(* PLC project Scenario_4b, Beckhoff Automation GmbH TwinCAT PLC Control 3.5.8.40 *)
(* stored: creationDateTime 2017-07-24T10:06:21.7701888, modificationDateTime 2017-07-24T10:06:21.774189 *)

PROGRAM MAIN
                                            VAR
                                            PPU : PPU;

                                            //WPType
                                            //Stack WPType
                                            Stack_WPType_Black : BOOL;
                                            Stack_WPType_White : BOOL;
                                            Stack_WPType_Metallic : BOOL;
                                            //Crane WPType
                                            Crane_WPType_Black : BOOL;
                                            Crane_WPType_White : BOOL;
                                            Crane_WPType_Metallic : BOOL;
                                            //Stamp WPType
                                            Stamp_WPType_Black : BOOL;
                                            Stamp_WPType_White : BOOL;
                                            Stamp_WPType_Metallic : BOOL;

                                            //Free Signale for follow plant section
                                            //Stack
                                            Stack_WPProvided : BOOL;
                                            //Crane
                                            Crane_Allow_Stamp_to_Operate : BOOL;
                                            Crane_PickedUpStackWP : BOOL;
                                            //Stamp
                                            Stamp_IsStamping : BOOL;
                                            Stamp_WPAvailable : BOOL;
                                            Stamp_AutomaticExecuteCompleted : BOOL;

                                            END_VAR

                                    PPU();
                                        PPU.Stack();
                                        PPU.Crane();
                                        PPU.Stamp();


                                        //WPType
                                        //Stack WPType
                                        Stack_WPType_Black := PPU.Stack.WPType_Black;
                                        Stack_WPType_Metallic := PPU.Stack.WPType_Metallic;
                                        //Crane WPType
                                        Crane_WPType_Black := PPU.Crane.WPType_Black;
                                        Crane_WPType_Metallic := PPU.Crane.WPType_Metallic;
                                        //Stamp WPType
                                        Stamp_WPType_Black := PPU.Stamp.WPType_Black;
                                        Stamp_WPType_Metallic := PPU.Stamp.WPType_Metallic;

                                        //Free Signale for follow plant section
                                        //Stack
                                        Stack_WPProvided := PPU.Stack.WPProvided;
                                        //Crane
                                        Crane_Allow_Stamp_to_Operate := PPU.Crane.Stamp_AllowedToOperate;
                                        Crane_PickedUpStackWP := PPU.Crane.Table.AtStack.DI_SwitchTrue AND
                                        PPU.Crane.WPPickedUp;
                                        //Stamp
                                        Stamp_IsStamping := PPU.Stamp.IsStamping;
                                        Stamp_WPAvailable := PPU.Stamp.WPAvailable.DI_SwitchTrue;
                                        Stamp_AutomaticExecuteCompleted := PPU.Stamp.AutomaticExecuteCompleted;
                                    
                                
END_PROGRAM

FUNCTION_BLOCK BistableCylinder
                                            VAR_INPUT
                                            END_VAR
                                            VAR_OUTPUT
                                            //Software
                                            Extended : BOOL;
                                            Retracted : BOOL;
                                            END_VAR
                                            VAR
                                            //Hardware
                                            DI_Extended AT %I* : BOOL;
                                            DI_Retracted AT %I* : BOOL;
                                            DO_Extend AT %Q* : BOOL;
                                            DO_Retract AT %Q* : BOOL;
                                            END_VAR

                                    
                                

ACTION ACT_Extend:
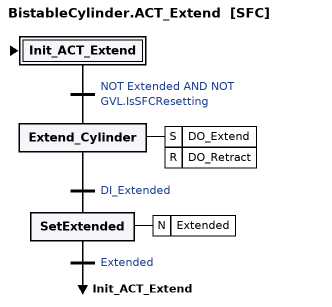
INITIAL_STEP Init_ACT_Extend:
END_STEP
TRANSITION FROM Init_ACT_Extend TO Extend_Cylinder
  := NOT Extended AND NOT GVL.IsSFCResetting;
END_TRANSITION
STEP Extend_Cylinder:
  DO_Extend(S);
  DO_Retract(R);
END_STEP
TRANSITION FROM Extend_Cylinder TO SetExtended
  := DI_Extended;
END_TRANSITION
STEP SetExtended:
  Extended(N);
END_STEP
TRANSITION FROM SetExtended TO Init_ACT_Extend
  := Extended;
END_TRANSITION
END_ACTION

ACTION ACT_Retract:
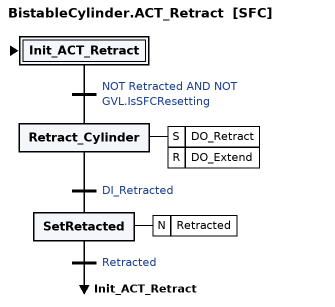
INITIAL_STEP Init_ACT_Retract:
END_STEP
TRANSITION FROM Init_ACT_Retract TO Retract_Cylinder
  := NOT Retracted AND NOT GVL.IsSFCResetting;
END_TRANSITION
STEP Retract_Cylinder:
  DO_Retract(S);
  DO_Extend(R);
END_STEP
TRANSITION FROM Retract_Cylinder TO SetRetacted
  := DI_Retracted;
END_TRANSITION
STEP SetRetacted:
  Retracted(N);
END_STEP
TRANSITION FROM SetRetacted TO Init_ACT_Retract
  := Retracted;
END_TRANSITION
END_ACTION
END_FUNCTION_BLOCK

FUNCTION_BLOCK InductiveSensor
                                            VAR_INPUT
                                            END_VAR
                                            VAR_OUTPUT
                                            END_VAR
                                            VAR
                                            //Hardware
                                            DI_WPMetallic AT %I* : BOOL;
                                            END_VAR

                                    
                                
END_FUNCTION_BLOCK

FUNCTION_BLOCK MicroSwitch
                                            VAR_INPUT
                                            END_VAR
                                            VAR_OUTPUT
                                            END_VAR
                                            VAR
                                            //Hardware
                                            DI_SwitchTrue AT %I* : BOOL;
                                            END_VAR

                                    
                                
END_FUNCTION_BLOCK

FUNCTION_BLOCK InductiveSwitch
                                            VAR_INPUT
                                            END_VAR
                                            VAR_OUTPUT
                                            END_VAR
                                            VAR
                                            //Hardware
                                            DI_InductiveSwitchTrue AT %I* : BOOL;
                                            END_VAR

                                    
                                
END_FUNCTION_BLOCK

FUNCTION_BLOCK MonostableCylinder
                                            VAR_INPUT
                                            END_VAR
                                            VAR_OUTPUT
                                            //Software
                                            Extended : BOOL;
                                            Retracted : BOOL;
                                            END_VAR
                                            VAR
                                            //Hardware
                                            DI_Extended AT %I* : BOOL;
                                            DI_Retracted AT %I* : BOOL;
                                            DO_Extend AT %Q* : BOOL;
                                            END_VAR

                                    
                                

ACTION ACT_Extend:
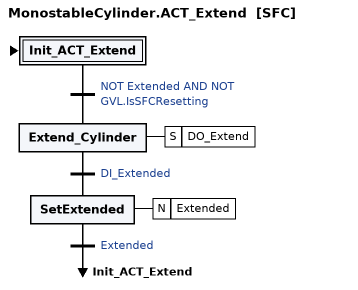
INITIAL_STEP Init_ACT_Extend:
END_STEP
TRANSITION FROM Init_ACT_Extend TO Extend_Cylinder
  := NOT Extended AND NOT GVL.IsSFCResetting;
END_TRANSITION
STEP Extend_Cylinder:
  DO_Extend(S);
END_STEP
TRANSITION FROM Extend_Cylinder TO SetExtended
  := DI_Extended;
END_TRANSITION
STEP SetExtended:
  Extended(N);
END_STEP
TRANSITION FROM SetExtended TO Init_ACT_Extend
  := Extended;
END_TRANSITION
END_ACTION

ACTION ACT_Retract:
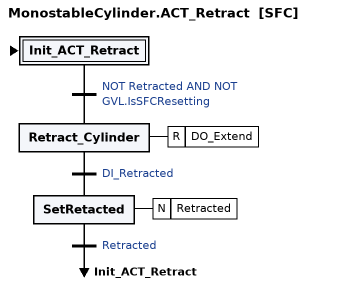
INITIAL_STEP Init_ACT_Retract:
END_STEP
TRANSITION FROM Init_ACT_Retract TO Retract_Cylinder
  := NOT Retracted AND NOT GVL.IsSFCResetting;
END_TRANSITION
STEP Retract_Cylinder:
  DO_Extend(R);
END_STEP
TRANSITION FROM Retract_Cylinder TO SetRetacted
  := DI_Retracted;
END_TRANSITION
STEP SetRetacted:
  Retracted(N);
END_STEP
TRANSITION FROM SetRetacted TO Init_ACT_Retract
  := Retracted;
END_TRANSITION
END_ACTION
END_FUNCTION_BLOCK

FUNCTION_BLOCK Motor
                                            VAR_INPUT
                                            END_VAR
                                            VAR_OUTPUT
                                            //Software
                                            Stopped : BOOL;
                                            TurningClockwise : BOOL;
                                            TurningCounterclockwise : BOOL;
                                            END_VAR
                                            VAR
                                            //Hardware
                                            DO_TurnClockwise AT %Q* : BOOL;
                                            DO_TurnCounterclockwise AT %Q* : BOOL;
                                            END_VAR

                                    
                                

ACTION ACT_Stop:
                                            DO_TurnClockwise := FALSE;
                                                DO_TurnCounterclockwise := FALSE;

                                                Stopped := TRUE;
                                                TurningClockwise := FALSE;
                                                TurningCounterclockwise := FALSE;
                                            
                                        
END_ACTION

ACTION ACT_TurnClockwise:
                                            DO_TurnClockwise := TRUE;
                                                DO_TurnCounterclockwise := FALSE;

                                                Stopped := FALSE;
                                                TurningClockwise := TRUE;
                                                TurningCounterclockwise := FALSE;
                                            
                                        
END_ACTION

ACTION ACT_TurnCounterclockwise:
                                            DO_TurnClockwise := FALSE;
                                                DO_TurnCounterclockwise := TRUE;

                                                Stopped := FALSE;
                                                TurningClockwise := FALSE;
                                                TurningCounterclockwise := TRUE;
                                            
                                        
END_ACTION
END_FUNCTION_BLOCK

FUNCTION_BLOCK OperationPanel
                                            VAR_INPUT
                                            END_VAR
                                            VAR_OUTPUT
                                            //Software
                                            EmergencyStop : BOOL;
                                            StartButton : BOOL;
                                            ManuelMode : BOOL;
                                            END_VAR
                                            VAR
                                            //Hardware
                                            DI_StartButton AT %I* : BOOL;
                                            DI_ManuelButton AT %I* : BOOL;
                                            DI_EmergencyStop AT %I* : BOOL;
                                            DO_LampGreen AT %Q* : BOOL;
                                            DO_LampWhite AT %Q* : BOOL;
                                            END_VAR

                                    EmergencyStop := NOT DI_EmergencyStop;
                                        StartButton := DI_StartButton;
                                        ManuelMode := DI_ManuelButton;
                                    
                                

ACTION ACT_TurnLampGreen_Off:
                                            DO_LampGreen := FALSE;
                                        
END_ACTION

ACTION ACT_TurnLampGreen_On:
                                            DO_LampGreen := TRUE;
                                        
END_ACTION

ACTION ACT_TurnLampWhite_Off:
                                            DO_LampWhite:=FALSE;
                                        
END_ACTION

ACTION ACT_TurnLampWhite_On:
                                            DO_LampWhite:=TRUE;
                                        
END_ACTION
END_FUNCTION_BLOCK

FUNCTION_BLOCK ProportionalValve
                                            VAR_INPUT
                                            //Hardware
                                            AO_SetPressure AT %Q* : INT;
                                            END_VAR
                                            VAR_OUTPUT
                                            END_VAR
                                            VAR
                                            END_VAR

                                    
                                
END_FUNCTION_BLOCK

FUNCTION_BLOCK TurningTable
                                            VAR_INPUT
                                            END_VAR
                                            VAR_OUTPUT
                                            END_VAR
                                            VAR
                                            //Hardware
                                            Motor : Motor;
                                            AtStack : MicroSwitch;
                                            AtRamp : MicroSwitch;
                                            AtStamp : MicroSwitch;
                                            AtStackInd : InductiveSwitch;
                                            AtRampInd : InductiveSwitch;
                                            AtStampInd : InductiveSwitch;

                                            END_VAR

                                    
                                
END_FUNCTION_BLOCK

FUNCTION_BLOCK VacuumGripper
                                            VAR_INPUT
                                            //Hardware
                                            Valve : Valve;
                                            VacuumSwitch : VacuumSwitch;
                                            END_VAR
                                            VAR_OUTPUT
                                            //Software
                                            Intaken : BOOL;
                                            Released : BOOL;
                                            END_VAR
                                            VAR
                                            END_VAR

                                    
                                

ACTION ACT_Intake:
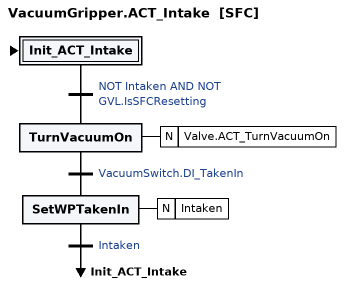
INITIAL_STEP Init_ACT_Intake:
END_STEP
TRANSITION FROM Init_ACT_Intake TO TurnVacuumOn
  := NOT Intaken AND NOT GVL.IsSFCResetting;
END_TRANSITION
STEP TurnVacuumOn:
  Valve.ACT_TurnVacuumOn(N);
END_STEP
TRANSITION FROM TurnVacuumOn TO SetWPTakenIn
  := VacuumSwitch.DI_TakenIn;
END_TRANSITION
STEP SetWPTakenIn:
  Intaken(N);
END_STEP
TRANSITION FROM SetWPTakenIn TO Init_ACT_Intake
  := Intaken;
END_TRANSITION
END_ACTION

ACTION ACT_Release:
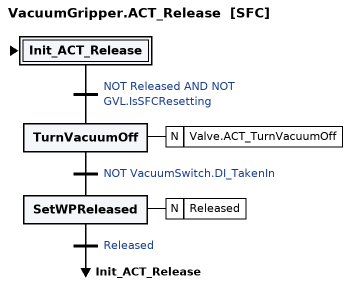
INITIAL_STEP Init_ACT_Release:
END_STEP
TRANSITION FROM Init_ACT_Release TO TurnVacuumOff
  := NOT Released AND NOT GVL.IsSFCResetting;
END_TRANSITION
STEP TurnVacuumOff:
  Valve.ACT_TurnVacuumOff(N);
END_STEP
TRANSITION FROM TurnVacuumOff TO SetWPReleased
  := NOT VacuumSwitch.DI_TakenIn;
END_TRANSITION
STEP SetWPReleased:
  Released(N);
END_STEP
TRANSITION FROM SetWPReleased TO Init_ACT_Release
  := Released;
END_TRANSITION
END_ACTION
END_FUNCTION_BLOCK

FUNCTION_BLOCK VacuumSwitch
                                            VAR_INPUT
                                            END_VAR
                                            VAR_OUTPUT
                                            END_VAR
                                            VAR
                                            //Hardware
                                            DI_TakenIn AT %I* : BOOL;
                                            END_VAR

                                    
                                
END_FUNCTION_BLOCK

FUNCTION_BLOCK Valve
                                            VAR_INPUT
                                            END_VAR
                                            VAR_OUTPUT
                                            END_VAR
                                            VAR
                                            //Hardware
                                            DO_VacuumOn AT %Q* : BOOL;
                                            END_VAR

                                    
                                

ACTION ACT_TurnVacuumOff:
                                            DO_VacuumOn := FALSE;
                                        
END_ACTION

ACTION ACT_TurnVacuumOn:
                                            DO_VacuumOn := TRUE;
                                        
END_ACTION
END_FUNCTION_BLOCK

FUNCTION_BLOCK Crane
                                            VAR_INPUT
                                            //Hardware
                                            LiftingCylinder : MonostableCylinder;
                                            Gripper : VacuumGripper;
                                            Table : TurningTable;
                                            //Software
                                            InitCompleted : BOOL;
                                            AutomaticExecuteCompleted : BOOL;
                                            Stamp_AllowedToOperate : BOOL;
                                            Stamp_WPStamped : BOOL;
                                            SoftwareEmergency : BOOL;
                                            EmergencyHandled : BOOL;
                                            SFCReset : BOOL; //Only for SFC implementation
                                            END_VAR
                                            VAR_OUTPUT
                                            //Software
                                            WPPickedUp : BOOL;
                                            WPPutDown : BOOL;
                                            ReachedStack : BOOL;
                                            ReachedRamp : BOOL;
                                            ReachedStamp : BOOL;
                                            WPType_Black : BOOL;
                                            WPType_Metallic : BOOL;
                                            END_VAR
                                            VAR
                                            //Hardware
                                            CraneSpeed AT %Q* : INT;

                                            //Software
                                            Timer : TON;
                                            Check_Stack_WPProvided : BOOL;
                                            Check_Stack_WPType_Black : BOOL;
                                            Check_Stack_WPType_Metallic : BOOL;
                                            Check_Stamp_IsStamping : BOOL;
                                            Check_Stamp_WPAvailable : BOOL;
                                            Check_Stamp_AutomaticExecuteCompleted : BOOL;
                                            END_VAR

                                    Check_Stack_WPProvided :=
                                        Main.Stack_WPProvided;
                                        Check_Stack_WPType_Black := Main.Stack_WPType_Black;
                                        Check_Stack_WPType_Metallic := Main.Stack_WPType_Metallic;
                                        Check_Stamp_IsStamping := Main.Stamp_IsStamping;
                                        Check_Stamp_WPAvailable := Main.Stamp_WPAvailable;
                                        Check_Stamp_AutomaticExecuteCompleted := Main.Stamp_AutomaticExecuteCompleted;
                                    
                                

ACTION Reset_StampAllowedToOperate:
                                            Stamp_AllowedToOperate :=
                                                FALSE;
                                            
                                        
END_ACTION

ACTION Reset_Timer:
                                            Timer(IN:=FALSE);
                                        
END_ACTION

ACTION Reset_Variables:
                                            InitCompleted := FALSE;
                                                AutomaticExecuteCompleted := FALSE;
                                                Stamp_AllowedToOperate := FALSE;

                                                WPPickedUp := FALSE;
                                                WPPutDown := FALSE;
                                                ReachedStack := FALSE;
                                                ReachedRamp := FALSE;
                                                ReachedStamp := FALSE;
                                                WPType_Black := FALSE;
                                                WPType_Metallic := FALSE;
                                            
                                        
END_ACTION

ACTION Set_StampAllowedToOperate:
                                            Stamp_AllowedToOperate :=
                                                TRUE;
                                            
                                        
END_ACTION

ACTION Set_Timer50ms:
                                            Timer(IN:=TRUE, PT:=T#50MS);
                                            
                                        
END_ACTION

ACTION Set_WPTypeEqualsStack:
                                            
                                                WPType_Black:=Main.Stack_WPType_Black;
                                                WPType_Metallic:=Main.Stack_WPType_Metallic;
                                            
                                        
END_ACTION

ACTION Set_WPTypeEqualsStamp:
                                            
                                                WPType_Black:=Main.Stamp_WPType_Black;
                                                WPType_Metallic:=Main.Stamp_WPType_Metallic;
                                            
                                        
END_ACTION

ACTION TurnClockwise_AND_Timer8000ms:
                                            Table.Motor.ACT_TurnClockwise();
                                                Timer(IN:=TRUE, PT:=T#8000MS);
                                            
                                        
END_ACTION

ACTION TurnCounterclockwise_AND_Timer8000ms:
                                            
                                                Table.Motor.ACT_TurnCounterclockwise();
                                                Timer(IN:=TRUE, PT:=T#8000MS);
                                            
                                        
END_ACTION

ACTION TurnVacuumOn_AND_Timer2000ms:
                                            Gripper.ACT_Intake();
                                                Timer(IN:=TRUE, PT:=T#2000MS);
                                            
                                        
END_ACTION

ACTION ACT_MoveToRamp:
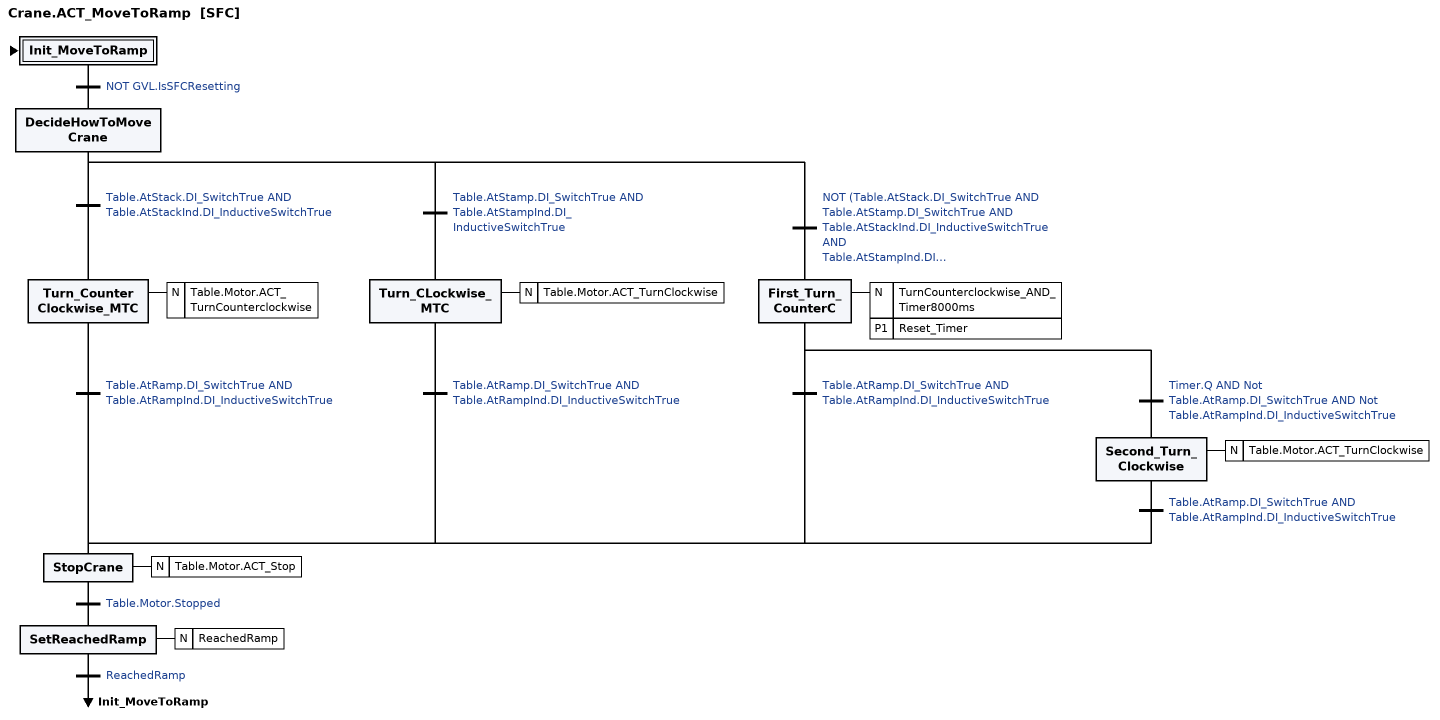
INITIAL_STEP Init_MoveToRamp:
END_STEP
TRANSITION FROM Init_MoveToRamp TO DecideHowToMoveCrane
  := NOT GVL.IsSFCResetting;
END_TRANSITION
STEP DecideHowToMoveCrane:
END_STEP
TRANSITION FROM DecideHowToMoveCrane TO Turn_CounterClockwise_MTC
  := Table.AtStack.DI_SwitchTrue AND
                                                    Table.AtStackInd.DI_InductiveSwitchTrue;
END_TRANSITION
TRANSITION FROM DecideHowToMoveCrane TO Turn_CLockwise_MTC
  := Table.AtStamp.DI_SwitchTrue AND
                                                    Table.AtStampInd.DI_InductiveSwitchTrue;
END_TRANSITION
TRANSITION FROM DecideHowToMoveCrane TO First_Turn_CounterC
  := NOT (Table.AtStack.DI_SwitchTrue AND
                                                    Table.AtStamp.DI_SwitchTrue AND
                                                    Table.AtStackInd.DI_InductiveSwitchTrue AND
                                                    Table.AtStampInd.DI_InductiveSwitchTrue);
END_TRANSITION
STEP Turn_CounterClockwise_MTC:
  Table.Motor.ACT_TurnCounterclockwise(N);
END_STEP
TRANSITION FROM Turn_CounterClockwise_MTC TO StopCrane
  := Table.AtRamp.DI_SwitchTrue AND
                                                    Table.AtRampInd.DI_InductiveSwitchTrue;
END_TRANSITION
STEP Turn_CLockwise_MTC:
  Table.Motor.ACT_TurnClockwise(N);
END_STEP
TRANSITION FROM Turn_CLockwise_MTC TO StopCrane
  := Table.AtRamp.DI_SwitchTrue AND
                                                    Table.AtRampInd.DI_InductiveSwitchTrue;
END_TRANSITION
STEP First_Turn_CounterC:
  TurnCounterclockwise_AND_Timer8000ms(N);
  Reset_Timer(P1);
END_STEP
TRANSITION FROM First_Turn_CounterC TO StopCrane
  := Table.AtRamp.DI_SwitchTrue AND
                                                    Table.AtRampInd.DI_InductiveSwitchTrue;
END_TRANSITION
TRANSITION FROM First_Turn_CounterC TO Second_Turn_Clockwise
  := Timer.Q AND Not Table.AtRamp.DI_SwitchTrue AND Not
                                                    Table.AtRampInd.DI_InductiveSwitchTrue;
END_TRANSITION
STEP Second_Turn_Clockwise:
  Table.Motor.ACT_TurnClockwise(N);
END_STEP
TRANSITION FROM Second_Turn_Clockwise TO StopCrane
  := Table.AtRamp.DI_SwitchTrue AND
                                                    Table.AtRampInd.DI_InductiveSwitchTrue;
END_TRANSITION
STEP StopCrane:
  Table.Motor.ACT_Stop(N);
END_STEP
TRANSITION FROM StopCrane TO SetReachedRamp
  := Table.Motor.Stopped;
END_TRANSITION
STEP SetReachedRamp:
  ReachedRamp(N);
END_STEP
TRANSITION FROM SetReachedRamp TO Init_MoveToRamp
  := ReachedRamp;
END_TRANSITION
END_ACTION

ACTION ACT_MoveToStack:
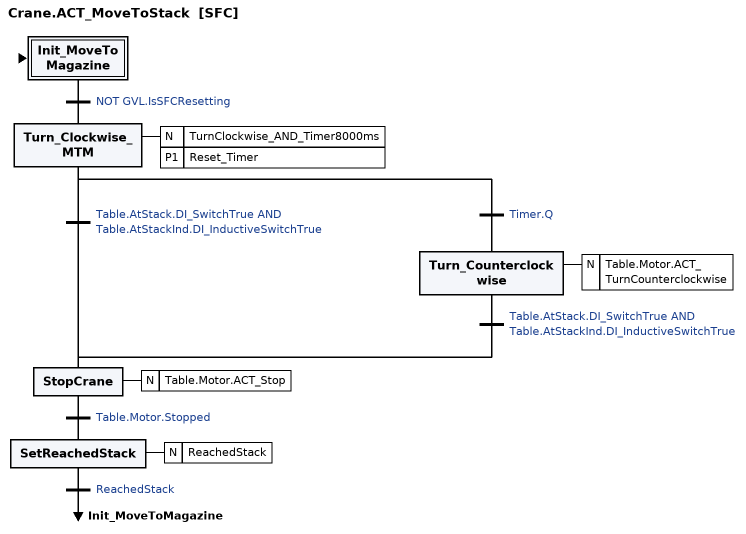
INITIAL_STEP Init_MoveToMagazine:
END_STEP
TRANSITION FROM Init_MoveToMagazine TO Turn_Clockwise_MTM
  := NOT GVL.IsSFCResetting;
END_TRANSITION
STEP Turn_Clockwise_MTM:
  TurnClockwise_AND_Timer8000ms(N);
  Reset_Timer(P1);
END_STEP
TRANSITION FROM Turn_Clockwise_MTM TO StopCrane
  := Table.AtStack.DI_SwitchTrue AND
                                                    Table.AtStackInd.DI_InductiveSwitchTrue;
END_TRANSITION
TRANSITION FROM Turn_Clockwise_MTM TO Turn_Counterclockwise
  := Timer.Q;
END_TRANSITION
STEP Turn_Counterclockwise:
  Table.Motor.ACT_TurnCounterclockwise(N);
END_STEP
TRANSITION FROM Turn_Counterclockwise TO StopCrane
  := Table.AtStack.DI_SwitchTrue AND
                                                    Table.AtStackInd.DI_InductiveSwitchTrue;
END_TRANSITION
STEP StopCrane:
  Table.Motor.ACT_Stop(N);
END_STEP
TRANSITION FROM StopCrane TO SetReachedStack
  := Table.Motor.Stopped;
END_TRANSITION
STEP SetReachedStack:
  ReachedStack(N);
END_STEP
TRANSITION FROM SetReachedStack TO Init_MoveToMagazine
  := ReachedStack;
END_TRANSITION
END_ACTION

ACTION ACT_MoveToStamp:
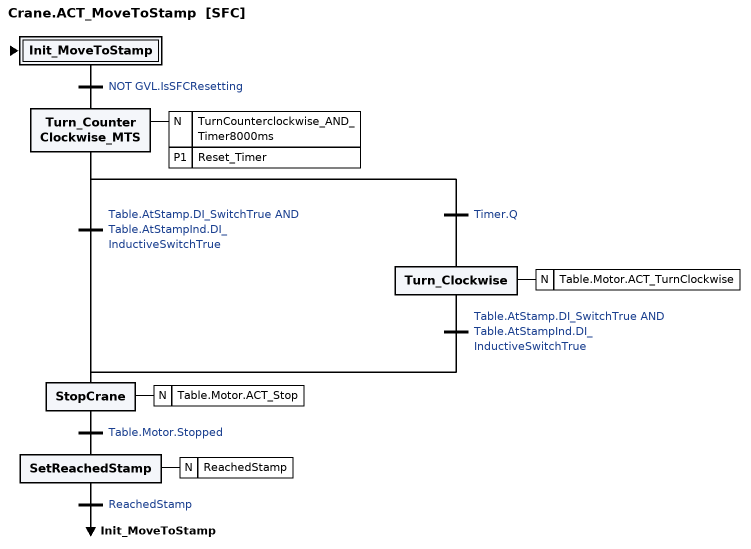
INITIAL_STEP Init_MoveToStamp:
END_STEP
TRANSITION FROM Init_MoveToStamp TO Turn_CounterClockwise_MTS
  := NOT GVL.IsSFCResetting;
END_TRANSITION
STEP Turn_CounterClockwise_MTS:
  TurnCounterclockwise_AND_Timer8000ms(N);
  Reset_Timer(P1);
END_STEP
TRANSITION FROM Turn_CounterClockwise_MTS TO StopCrane
  := Table.AtStamp.DI_SwitchTrue AND
                                                    Table.AtStampInd.DI_InductiveSwitchTrue;
END_TRANSITION
TRANSITION FROM Turn_CounterClockwise_MTS TO Turn_Clockwise
  := Timer.Q;
END_TRANSITION
STEP Turn_Clockwise:
  Table.Motor.ACT_TurnClockwise(N);
END_STEP
TRANSITION FROM Turn_Clockwise TO StopCrane
  := Table.AtStamp.DI_SwitchTrue AND
                                                    Table.AtStampInd.DI_InductiveSwitchTrue;
END_TRANSITION
STEP StopCrane:
  Table.Motor.ACT_Stop(N);
END_STEP
TRANSITION FROM StopCrane TO SetReachedStamp
  := Table.Motor.Stopped;
END_TRANSITION
STEP SetReachedStamp:
  ReachedStamp(N);
END_STEP
TRANSITION FROM SetReachedStamp TO Init_MoveToStamp
  := ReachedStamp;
END_TRANSITION
END_ACTION

ACTION ACT_PickUpWP:
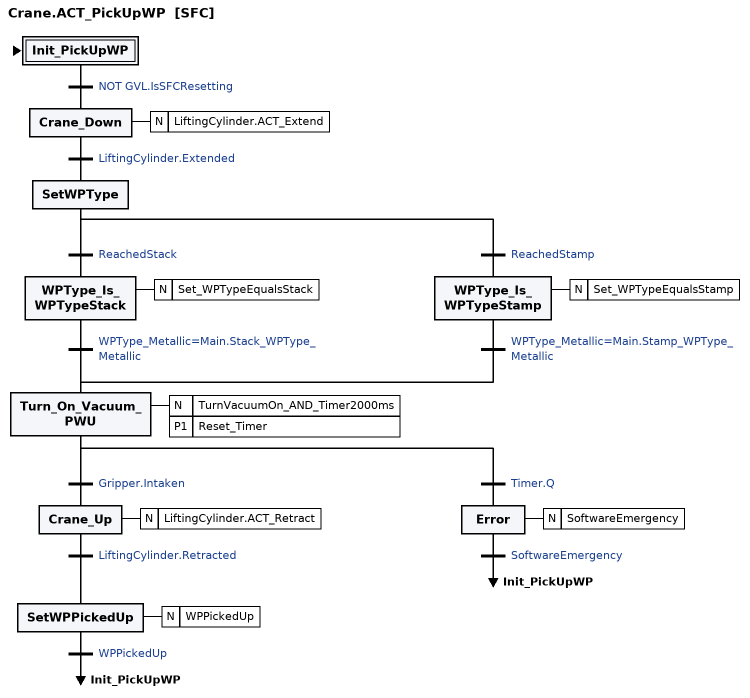
INITIAL_STEP Init_PickUpWP:
END_STEP
TRANSITION FROM Init_PickUpWP TO Crane_Down
  := NOT GVL.IsSFCResetting;
END_TRANSITION
STEP Crane_Down:
  LiftingCylinder.ACT_Extend(N);
END_STEP
TRANSITION FROM Crane_Down TO SetWPType
  := LiftingCylinder.Extended;
END_TRANSITION
STEP SetWPType:
END_STEP
TRANSITION FROM SetWPType TO WPType_Is_WPTypeStack
  := ReachedStack;
END_TRANSITION
TRANSITION FROM SetWPType TO WPType_Is_WPTypeStamp
  := ReachedStamp;
END_TRANSITION
STEP WPType_Is_WPTypeStack:
  Set_WPTypeEqualsStack(N);
END_STEP
TRANSITION FROM WPType_Is_WPTypeStack TO Turn_On_Vacuum_PWU
  := WPType_Metallic=Main.Stack_WPType_Metallic;
END_TRANSITION
STEP WPType_Is_WPTypeStamp:
  Set_WPTypeEqualsStamp(N);
END_STEP
TRANSITION FROM WPType_Is_WPTypeStamp TO Turn_On_Vacuum_PWU
  := WPType_Metallic=Main.Stamp_WPType_Metallic;
END_TRANSITION
STEP Turn_On_Vacuum_PWU:
  TurnVacuumOn_AND_Timer2000ms(N);
  Reset_Timer(P1);
END_STEP
TRANSITION FROM Turn_On_Vacuum_PWU TO Crane_Up
  := Gripper.Intaken;
END_TRANSITION
TRANSITION FROM Turn_On_Vacuum_PWU TO Error
  := Timer.Q;
END_TRANSITION
STEP Crane_Up:
  LiftingCylinder.ACT_Retract(N);
END_STEP
TRANSITION FROM Crane_Up TO SetWPPickedUp
  := LiftingCylinder.Retracted;
END_TRANSITION
STEP Error:
  SoftwareEmergency(N);
END_STEP
TRANSITION FROM Error TO Init_PickUpWP
  := SoftwareEmergency;
END_TRANSITION
STEP SetWPPickedUp:
  WPPickedUp(N);
END_STEP
TRANSITION FROM SetWPPickedUp TO Init_PickUpWP
  := WPPickedUp;
END_TRANSITION
END_ACTION

ACTION ACT_PutDownWP:
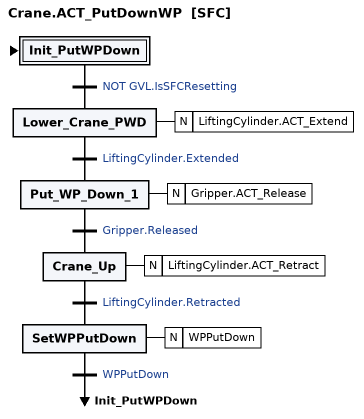
INITIAL_STEP Init_PutWPDown:
END_STEP
TRANSITION FROM Init_PutWPDown TO Lower_Crane_PWD
  := NOT GVL.IsSFCResetting;
END_TRANSITION
STEP Lower_Crane_PWD:
  LiftingCylinder.ACT_Extend(N);
END_STEP
TRANSITION FROM Lower_Crane_PWD TO Put_WP_Down_1
  := LiftingCylinder.Extended;
END_TRANSITION
STEP Put_WP_Down_1:
  Gripper.ACT_Release(N);
END_STEP
TRANSITION FROM Put_WP_Down_1 TO Crane_Up
  := Gripper.Released;
END_TRANSITION
STEP Crane_Up:
  LiftingCylinder.ACT_Retract(N);
END_STEP
TRANSITION FROM Crane_Up TO SetWPPutDown
  := LiftingCylinder.Retracted;
END_TRANSITION
STEP SetWPPutDown:
  WPPutDown(N);
END_STEP
TRANSITION FROM SetWPPutDown TO Init_PutWPDown
  := WPPutDown;
END_TRANSITION
END_ACTION

ACTION ACT_AutomaticExecute:
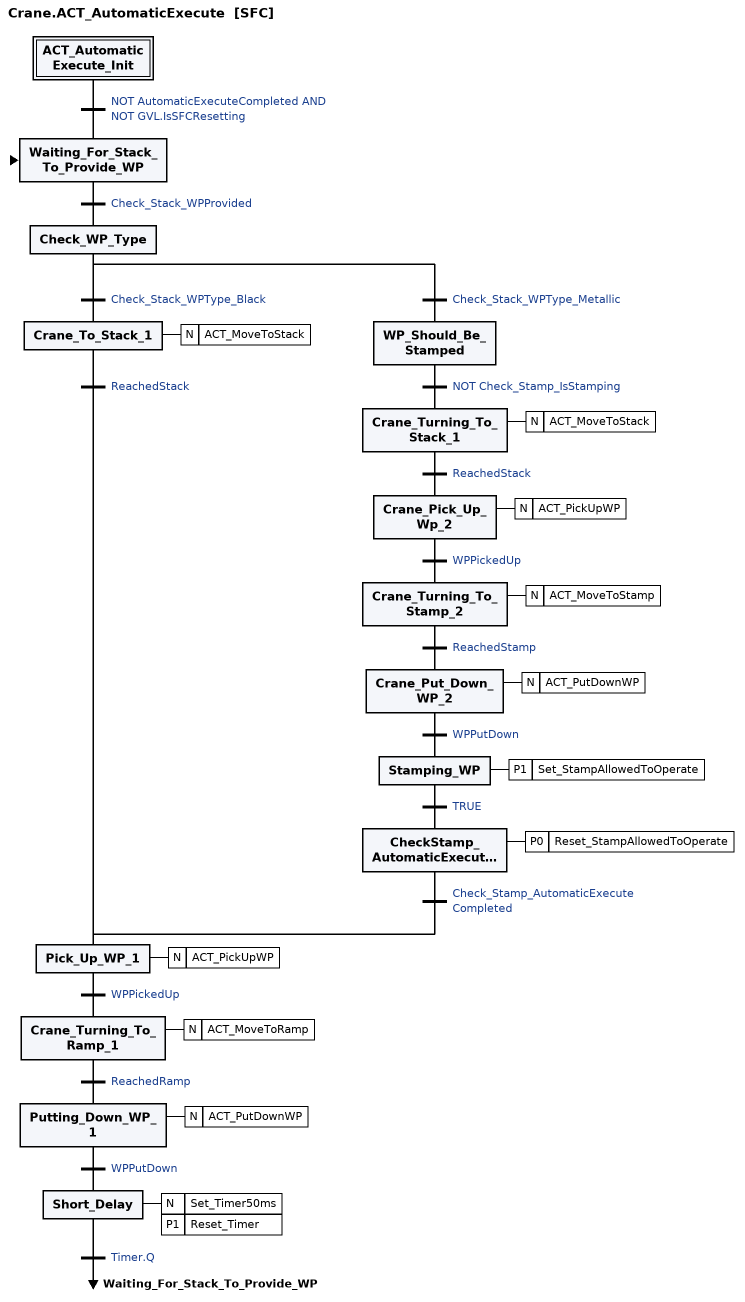
INITIAL_STEP ACT_AutomaticExecute_Init:
END_STEP
TRANSITION FROM ACT_AutomaticExecute_Init TO Waiting_For_Stack_To_Provide_WP
  := NOT AutomaticExecuteCompleted AND NOT GVL.IsSFCResetting;
END_TRANSITION
STEP Waiting_For_Stack_To_Provide_WP:
END_STEP
TRANSITION FROM Waiting_For_Stack_To_Provide_WP TO Check_WP_Type
  := Check_Stack_WPProvided;
END_TRANSITION
STEP Check_WP_Type:
END_STEP
TRANSITION FROM Check_WP_Type TO Crane_To_Stack_1
  := Check_Stack_WPType_Black;
END_TRANSITION
TRANSITION FROM Check_WP_Type TO WP_Should_Be_Stamped
  := Check_Stack_WPType_Metallic;
END_TRANSITION
STEP Crane_To_Stack_1:
  ACT_MoveToStack(N);
END_STEP
TRANSITION FROM Crane_To_Stack_1 TO Pick_Up_WP_1
  := ReachedStack;
END_TRANSITION
STEP Pick_Up_WP_1:
  ACT_PickUpWP(N);
END_STEP
TRANSITION FROM Pick_Up_WP_1 TO Crane_Turning_To_Ramp_1
  := WPPickedUp;
END_TRANSITION
STEP Crane_Turning_To_Ramp_1:
  ACT_MoveToRamp(N);
END_STEP
TRANSITION FROM Crane_Turning_To_Ramp_1 TO Putting_Down_WP_1
  := ReachedRamp;
END_TRANSITION
STEP Putting_Down_WP_1:
  ACT_PutDownWP(N);
END_STEP
TRANSITION FROM Putting_Down_WP_1 TO Short_Delay
  := WPPutDown;
END_TRANSITION
STEP Short_Delay:
  Set_Timer50ms(N);
  Reset_Timer(P1);
END_STEP
TRANSITION FROM Short_Delay TO Waiting_For_Stack_To_Provide_WP
  := Timer.Q;
END_TRANSITION
STEP WP_Should_Be_Stamped:
END_STEP
TRANSITION FROM WP_Should_Be_Stamped TO Crane_Turning_To_Stack_1
  := NOT Check_Stamp_IsStamping;
END_TRANSITION
STEP Crane_Turning_To_Stack_1:
  ACT_MoveToStack(N);
END_STEP
TRANSITION FROM Crane_Turning_To_Stack_1 TO Crane_Pick_Up_Wp_2
  := ReachedStack;
END_TRANSITION
STEP Crane_Pick_Up_Wp_2:
  ACT_PickUpWP(N);
END_STEP
TRANSITION FROM Crane_Pick_Up_Wp_2 TO Crane_Turning_To_Stamp_2
  := WPPickedUp;
END_TRANSITION
STEP Crane_Turning_To_Stamp_2:
  ACT_MoveToStamp(N);
END_STEP
TRANSITION FROM Crane_Turning_To_Stamp_2 TO Crane_Put_Down_WP_2
  := ReachedStamp;
END_TRANSITION
STEP Crane_Put_Down_WP_2:
  ACT_PutDownWP(N);
END_STEP
TRANSITION FROM Crane_Put_Down_WP_2 TO Stamping_WP
  := WPPutDown;
END_TRANSITION
STEP Stamping_WP:
  Set_StampAllowedToOperate(P1);
END_STEP
TRANSITION FROM Stamping_WP TO CheckStamp_AutomaticExecuteCompleted
  := TRUE;
END_TRANSITION
STEP CheckStamp_AutomaticExecuteCompleted:
  Reset_StampAllowedToOperate(P0);
END_STEP
TRANSITION FROM CheckStamp_AutomaticExecuteCompleted TO Pick_Up_WP_1
  := Check_Stamp_AutomaticExecuteCompleted;
END_TRANSITION
END_ACTION

ACTION ACT_EmergencyStop:
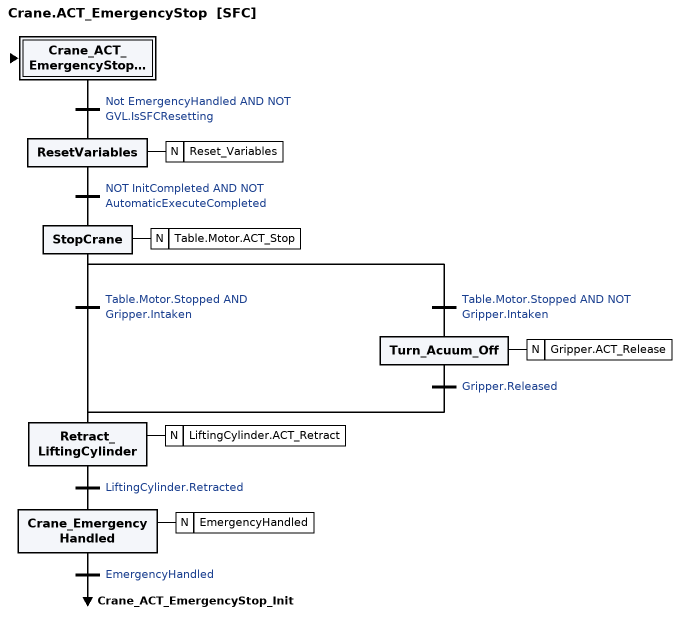
INITIAL_STEP Crane_ACT_EmergencyStop_Init:
END_STEP
TRANSITION FROM Crane_ACT_EmergencyStop_Init TO ResetVariables
  := Not EmergencyHandled AND NOT GVL.IsSFCResetting;
END_TRANSITION
STEP ResetVariables:
  Reset_Variables(N);
END_STEP
TRANSITION FROM ResetVariables TO StopCrane
  := NOT InitCompleted AND NOT AutomaticExecuteCompleted;
END_TRANSITION
STEP StopCrane:
  Table.Motor.ACT_Stop(N);
END_STEP
TRANSITION FROM StopCrane TO Retract_LiftingCylinder
  := Table.Motor.Stopped AND Gripper.Intaken;
END_TRANSITION
TRANSITION FROM StopCrane TO Turn_Acuum_Off
  := Table.Motor.Stopped AND NOT Gripper.Intaken;
END_TRANSITION
STEP Turn_Acuum_Off:
  Gripper.ACT_Release(N);
END_STEP
TRANSITION FROM Turn_Acuum_Off TO Retract_LiftingCylinder
  := Gripper.Released;
END_TRANSITION
STEP Retract_LiftingCylinder:
  LiftingCylinder.ACT_Retract(N);
END_STEP
TRANSITION FROM Retract_LiftingCylinder TO Crane_EmergencyHandled
  := LiftingCylinder.Retracted;
END_TRANSITION
STEP Crane_EmergencyHandled:
  EmergencyHandled(N);
END_STEP
TRANSITION FROM Crane_EmergencyHandled TO Crane_ACT_EmergencyStop_Init
  := EmergencyHandled;
END_TRANSITION
END_ACTION

ACTION ACT_Init:
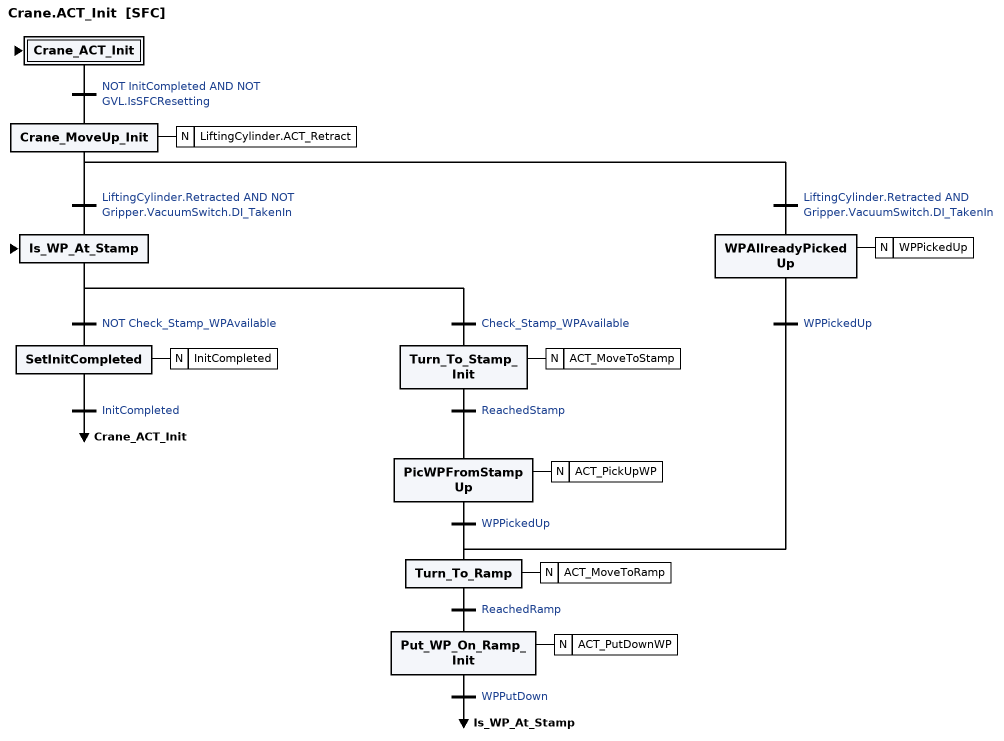
INITIAL_STEP Crane_ACT_Init:
END_STEP
TRANSITION FROM Crane_ACT_Init TO Crane_MoveUp_Init
  := NOT InitCompleted AND NOT GVL.IsSFCResetting;
END_TRANSITION
STEP Crane_MoveUp_Init:
  LiftingCylinder.ACT_Retract(N);
END_STEP
TRANSITION FROM Crane_MoveUp_Init TO Is_WP_At_Stamp
  := LiftingCylinder.Retracted AND NOT
                                                    Gripper.VacuumSwitch.DI_TakenIn;
END_TRANSITION
TRANSITION FROM Crane_MoveUp_Init TO WPAllreadyPickedUp
  := LiftingCylinder.Retracted AND
                                                    Gripper.VacuumSwitch.DI_TakenIn;
END_TRANSITION
STEP WPAllreadyPickedUp:
  WPPickedUp(N);
END_STEP
TRANSITION FROM WPAllreadyPickedUp TO Turn_To_Ramp
  := WPPickedUp;
END_TRANSITION
STEP Turn_To_Ramp:
  ACT_MoveToRamp(N);
END_STEP
TRANSITION FROM Turn_To_Ramp TO Put_WP_On_Ramp_Init
  := ReachedRamp;
END_TRANSITION
STEP Put_WP_On_Ramp_Init:
  ACT_PutDownWP(N);
END_STEP
TRANSITION FROM Put_WP_On_Ramp_Init TO Is_WP_At_Stamp
  := WPPutDown;
END_TRANSITION
STEP Is_WP_At_Stamp:
END_STEP
TRANSITION FROM Is_WP_At_Stamp TO SetInitCompleted
  := NOT Check_Stamp_WPAvailable;
END_TRANSITION
TRANSITION FROM Is_WP_At_Stamp TO Turn_To_Stamp_Init
  := Check_Stamp_WPAvailable;
END_TRANSITION
STEP Turn_To_Stamp_Init:
  ACT_MoveToStamp(N);
END_STEP
TRANSITION FROM Turn_To_Stamp_Init TO PicWPFromStampUp
  := ReachedStamp;
END_TRANSITION
STEP PicWPFromStampUp:
  ACT_PickUpWP(N);
END_STEP
TRANSITION FROM PicWPFromStampUp TO Turn_To_Ramp
  := WPPickedUp;
END_TRANSITION
STEP SetInitCompleted:
  InitCompleted(N);
END_STEP
TRANSITION FROM SetInitCompleted TO Crane_ACT_Init
  := InitCompleted;
END_TRANSITION
END_ACTION
END_FUNCTION_BLOCK

FUNCTION_BLOCK Stack
                                            VAR_INPUT
                                            //Hardware
                                            Seperator : MonostableCylinder;
                                            Panel : OperationPanel;
                                            WPAvailable : MicroSwitch;
                                            InductiveSensor : InductiveSensor;

                                            //Software
                                            StartButton : BOOL;
                                            InitCompleted : BOOL;
                                            AutomaticExecuteCompleted : BOOL;
                                            EmergencyStop : BOOL;
                                            EmergencyHandled : BOOL;
                                            SFCReset : BOOL; //Only for SFC implementation
                                            END_VAR
                                            VAR_OUTPUT
                                            //Software
                                            WPProvided : BOOL;
                                            WPType_Black : BOOL;
                                            WPType_Metallic : BOOL;
                                            END_VAR
                                            VAR
                                            //Software
                                            Timer : TON;
                                            Check_Crane_PickedUpWp : BOOL;
                                            END_VAR

                                    Panel();
                                        StartButton := Panel.StartButton;
                                        EmergencyStop := Panel.EmergencyStop;
                                        Check_Crane_PickedUpWP := Main.Crane_PickedUpStackWP;
                                    
                                

ACTION Reset_Timer:
                                            Timer(IN:=FALSE);
                                        
END_ACTION

ACTION Reset_Variables:
                                            InitCompleted := FALSE;
                                                AutomaticExecuteCompleted := FALSE;

                                                WPType_Black:=FALSE;
                                                WPType_Metallic:=FALSE;
                                            
                                        
END_ACTION

ACTION Set_Timer250ms:
                                            Timer(IN:=TRUE, PT:=T#250MS);
                                            
                                        
END_ACTION

ACTION Set_WPParameters_AND_WPProvided:
                                            IF(NOT
                                                InductiveSensor.DI_WPMetallic)THEN
                                                WPType_Black:=TRUE;
                                                WPType_Metallic:=FALSE;
                                                ELSIF(InductiveSensor.DI_WPMetallic)THEN
                                                WPType_Black:=FALSE;
                                                WPType_Metallic:=TRUE;
                                                END_IF

                                                WPProvided:=TRUE;
                                            
                                        
END_ACTION

ACTION ACT_ProvideWP:
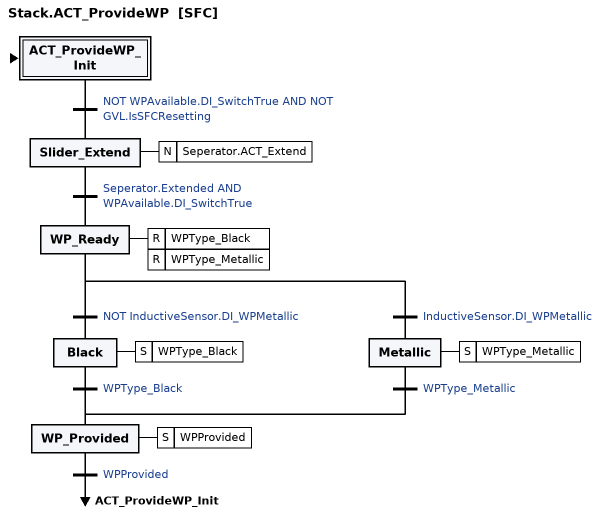
INITIAL_STEP ACT_ProvideWP_Init:
END_STEP
TRANSITION FROM ACT_ProvideWP_Init TO Slider_Extend
  := NOT WPAvailable.DI_SwitchTrue AND NOT GVL.IsSFCResetting;
END_TRANSITION
STEP Slider_Extend:
  Seperator.ACT_Extend(N);
END_STEP
TRANSITION FROM Slider_Extend TO WP_Ready
  := Seperator.Extended AND WPAvailable.DI_SwitchTrue;
END_TRANSITION
STEP WP_Ready:
  WPType_Black(R);
  WPType_Metallic(R);
END_STEP
TRANSITION FROM WP_Ready TO Black
  := NOT InductiveSensor.DI_WPMetallic;
END_TRANSITION
TRANSITION FROM WP_Ready TO Metallic
  := InductiveSensor.DI_WPMetallic;
END_TRANSITION
STEP Black:
  WPType_Black(S);
END_STEP
TRANSITION FROM Black TO WP_Provided
  := WPType_Black;
END_TRANSITION
STEP Metallic:
  WPType_Metallic(S);
END_STEP
TRANSITION FROM Metallic TO WP_Provided
  := WPType_Metallic;
END_TRANSITION
STEP WP_Provided:
  WPProvided(S);
END_STEP
TRANSITION FROM WP_Provided TO ACT_ProvideWP_Init
  := WPProvided;
END_TRANSITION
END_ACTION

ACTION ACT_AutomaticExecute:
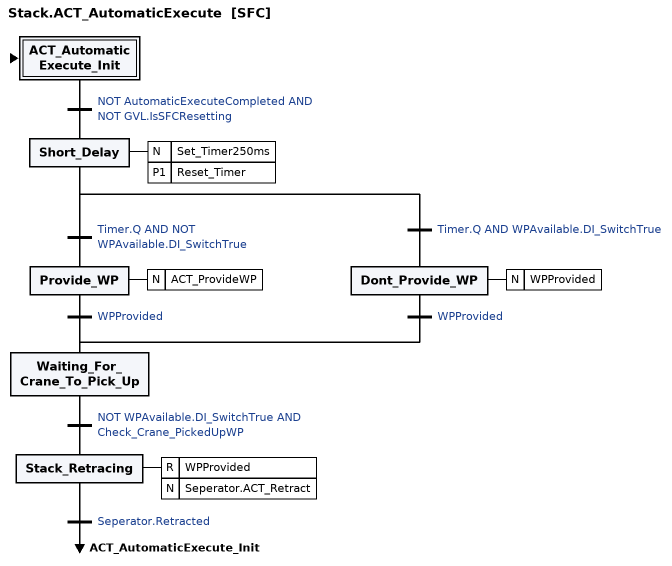
INITIAL_STEP ACT_AutomaticExecute_Init:
END_STEP
TRANSITION FROM ACT_AutomaticExecute_Init TO Short_Delay
  := NOT AutomaticExecuteCompleted AND NOT GVL.IsSFCResetting;
END_TRANSITION
STEP Short_Delay:
  Set_Timer250ms(N);
  Reset_Timer(P1);
END_STEP
TRANSITION FROM Short_Delay TO Provide_WP
  := Timer.Q AND NOT WPAvailable.DI_SwitchTrue;
END_TRANSITION
TRANSITION FROM Short_Delay TO Dont_Provide_WP
  := Timer.Q AND WPAvailable.DI_SwitchTrue;
END_TRANSITION
STEP Provide_WP:
  ACT_ProvideWP(N);
END_STEP
TRANSITION FROM Provide_WP TO Waiting_For_Crane_To_Pick_Up
  := WPProvided;
END_TRANSITION
STEP Dont_Provide_WP:
  WPProvided(N);
END_STEP
TRANSITION FROM Dont_Provide_WP TO Waiting_For_Crane_To_Pick_Up
  := WPProvided;
END_TRANSITION
STEP Waiting_For_Crane_To_Pick_Up:
END_STEP
TRANSITION FROM Waiting_For_Crane_To_Pick_Up TO Stack_Retracing
  := NOT WPAvailable.DI_SwitchTrue AND Check_Crane_PickedUpWP;
END_TRANSITION
STEP Stack_Retracing:
  WPProvided(R);
  Seperator.ACT_Retract(N);
END_STEP
TRANSITION FROM Stack_Retracing TO ACT_AutomaticExecute_Init
  := Seperator.Retracted;
END_TRANSITION
END_ACTION

ACTION ACT_EmergencyStop:
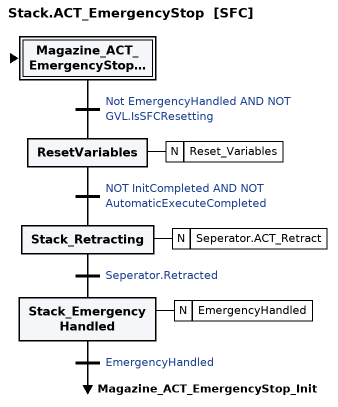
INITIAL_STEP Magazine_ACT_EmergencyStop_Init:
END_STEP
TRANSITION FROM Magazine_ACT_EmergencyStop_Init TO ResetVariables
  := Not EmergencyHandled AND NOT GVL.IsSFCResetting;
END_TRANSITION
STEP ResetVariables:
  Reset_Variables(N);
END_STEP
TRANSITION FROM ResetVariables TO Stack_Retracting
  := NOT InitCompleted AND NOT AutomaticExecuteCompleted;
END_TRANSITION
STEP Stack_Retracting:
  Seperator.ACT_Retract(N);
END_STEP
TRANSITION FROM Stack_Retracting TO Stack_EmergencyHandled
  := Seperator.Retracted;
END_TRANSITION
STEP Stack_EmergencyHandled:
  EmergencyHandled(N);
END_STEP
TRANSITION FROM Stack_EmergencyHandled TO Magazine_ACT_EmergencyStop_Init
  := EmergencyHandled;
END_TRANSITION
END_ACTION

ACTION ACT_Init:
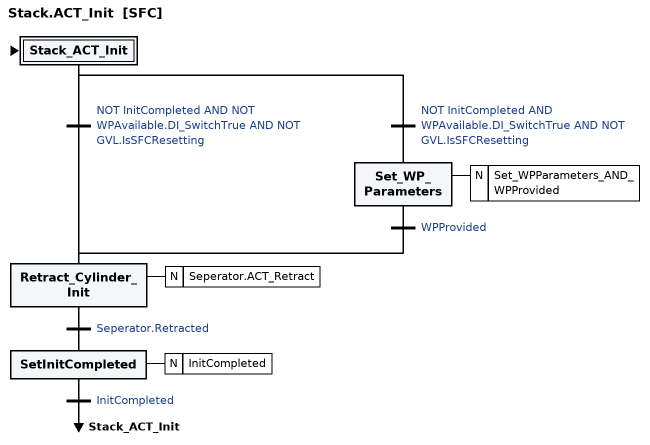
INITIAL_STEP Stack_ACT_Init:
END_STEP
TRANSITION FROM Stack_ACT_Init TO Retract_Cylinder_Init
  := NOT InitCompleted AND NOT WPAvailable.DI_SwitchTrue AND NOT
                                                    GVL.IsSFCResetting;
END_TRANSITION
TRANSITION FROM Stack_ACT_Init TO Set_WP_Parameters
  := NOT InitCompleted AND WPAvailable.DI_SwitchTrue AND NOT
                                                    GVL.IsSFCResetting;
END_TRANSITION
STEP Set_WP_Parameters:
  Set_WPParameters_AND_WPProvided(N);
END_STEP
TRANSITION FROM Set_WP_Parameters TO Retract_Cylinder_Init
  := WPProvided;
END_TRANSITION
STEP Retract_Cylinder_Init:
  Seperator.ACT_Retract(N);
END_STEP
TRANSITION FROM Retract_Cylinder_Init TO SetInitCompleted
  := Seperator.Retracted;
END_TRANSITION
STEP SetInitCompleted:
  InitCompleted(N);
END_STEP
TRANSITION FROM SetInitCompleted TO Stack_ACT_Init
  := InitCompleted;
END_TRANSITION
END_ACTION
END_FUNCTION_BLOCK

FUNCTION_BLOCK Stamp
                                            VAR_INPUT
                                            //Hardware
                                            Panel : OperationPanel;
                                            PropValve : ProportionalValve;
                                            WPAvailable : MicroSwitch;
                                            StampingCylinder : MonostableCylinder;
                                            SlidingCylinder : BistableCylinder;

                                            //Software
                                            StartButton : BOOL;
                                            InitCompleted : BOOL;
                                            AutomaticExecuteCompleted : BOOL;
                                            EmergencyStop : BOOL;
                                            SoftwareEmergency : BOOL;
                                            EmergencyHandled : BOOL;
                                            SFCReset : BOOL; //Only for SFC implementation
                                            END_VAR
                                            VAR_OUTPUT
                                            //Software
                                            IsStamping : BOOL;
                                            WPStamped : BOOL;
                                            WPType_Black : BOOL;
                                            WPType_Metallic : BOOL;
                                            END_VAR
                                            VAR
                                            //Software
                                            Timer : TON;
                                            Check_Allowed_To_Operate : BOOL;
                                            Check_WPType_Black : BOOL;
                                            Check_WPType_Metallic : BOOL;
                                            Check_Stamp_WPAvailable : BOOL;
                                            END_VAR

                                    Panel();
                                        StartButton := Panel.StartButton;
                                        EmergencyStop := Panel.EmergencyStop;
                                        Check_Allowed_To_Operate := Main.Crane_Allow_Stamp_to_Operate;
                                        Check_WPType_Black:=Main.Crane_WPType_Black;
                                        Check_WPType_Metallic:=Main.Crane_WPType_Metallic;
                                        Check_Stamp_WPAvailable:=Main.Stamp_WPAvailable;
                                    
                                

ACTION ExtendStampingCylinder_AND_Timer1500ms:
                                            StampingCylinder.ACT_Extend();
                                                Timer(IN:=TRUE, PT:=T#1500MS);
                                            
                                        
END_ACTION

ACTION Reset_Pressure:
                                            PropValve.AO_SetPressure:=0;
                                            
                                        
END_ACTION

ACTION Reset_Timer:
                                            Timer(IN:=FALSE);
                                        
END_ACTION

ACTION Reset_Variables:
                                            InitCompleted := FALSE;
                                                AutomaticExecuteCompleted := FALSE;

                                                propValve.AO_SetPressure:=0;
                                                IsStamping:=FALSE;
                                                WPStamped:=FALSE;
                                                WPType_Black := FALSE;
                                                WPType_Metallic := FALSE;
                                            
                                        
END_ACTION

ACTION Set_LightPressure:
                                            
                                                PropValve.AO_SetPressure:=4000;
                                            
                                        
END_ACTION

ACTION Set_Timer1000ms:
                                            Timer(IN:=TRUE, PT:=T#1000MS);
                                            
                                        
END_ACTION

ACTION Set_Timer500ms:
                                            Timer(IN:=TRUE, PT:=T#500ms);
                                            
                                        
END_ACTION

ACTION Set_WPType:
                                            WPType_Black :=
                                                Check_WPType_Black;
                                                WPType_Metallic := Check_WPType_Metallic;
                                            
                                        
END_ACTION

ACTION ACT_Stamp:
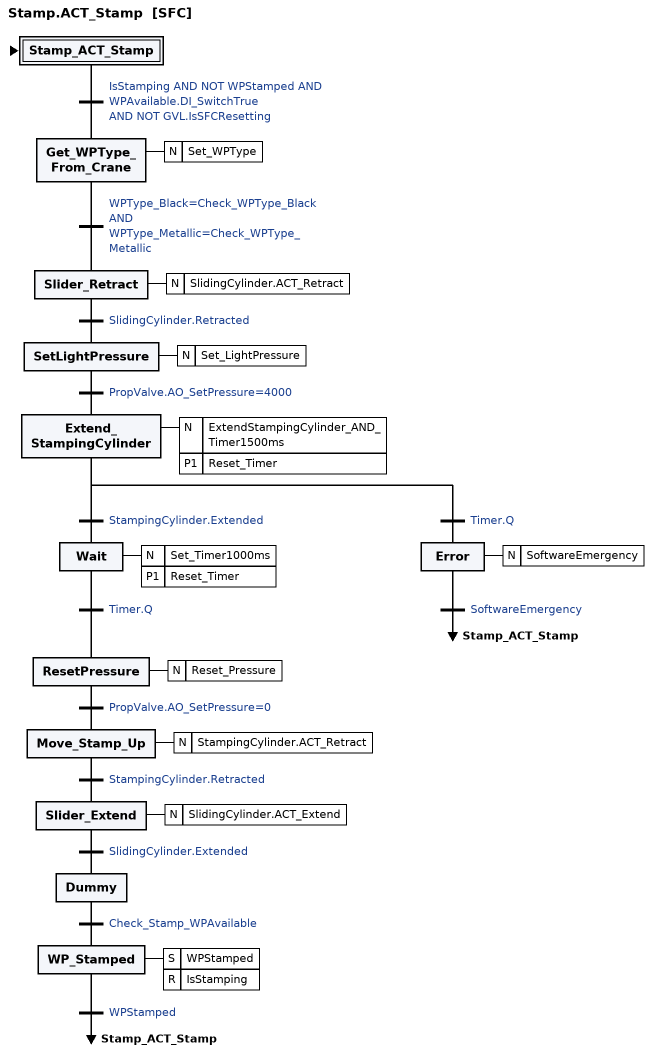
INITIAL_STEP Stamp_ACT_Stamp:
END_STEP
TRANSITION FROM Stamp_ACT_Stamp TO Get_WPType_From_Crane
  := IsStamping AND NOT WPStamped AND WPAvailable.DI_SwitchTrue
                                                    AND NOT GVL.IsSFCResetting;
END_TRANSITION
STEP Get_WPType_From_Crane:
  Set_WPType(N);
END_STEP
TRANSITION FROM Get_WPType_From_Crane TO Slider_Retract
  := WPType_Black=Check_WPType_Black AND
                                                    WPType_Metallic=Check_WPType_Metallic;
END_TRANSITION
STEP Slider_Retract:
  SlidingCylinder.ACT_Retract(N);
END_STEP
TRANSITION FROM Slider_Retract TO SetLightPressure
  := SlidingCylinder.Retracted;
END_TRANSITION
STEP SetLightPressure:
  Set_LightPressure(N);
END_STEP
TRANSITION FROM SetLightPressure TO Extend_StampingCylinder
  := PropValve.AO_SetPressure=4000;
END_TRANSITION
STEP Extend_StampingCylinder:
  ExtendStampingCylinder_AND_Timer1500ms(N);
  Reset_Timer(P1);
END_STEP
TRANSITION FROM Extend_StampingCylinder TO Wait
  := StampingCylinder.Extended;
END_TRANSITION
TRANSITION FROM Extend_StampingCylinder TO Error
  := Timer.Q;
END_TRANSITION
STEP Error:
  SoftwareEmergency(N);
END_STEP
TRANSITION FROM Error TO Stamp_ACT_Stamp
  := SoftwareEmergency;
END_TRANSITION
STEP Wait:
  Set_Timer1000ms(N);
  Reset_Timer(P1);
END_STEP
TRANSITION FROM Wait TO ResetPressure
  := Timer.Q;
END_TRANSITION
STEP ResetPressure:
  Reset_Pressure(N);
END_STEP
TRANSITION FROM ResetPressure TO Move_Stamp_Up
  := PropValve.AO_SetPressure=0;
END_TRANSITION
STEP Move_Stamp_Up:
  StampingCylinder.ACT_Retract(N);
END_STEP
TRANSITION FROM Move_Stamp_Up TO Slider_Extend
  := StampingCylinder.Retracted;
END_TRANSITION
STEP Slider_Extend:
  SlidingCylinder.ACT_Extend(N);
END_STEP
TRANSITION FROM Slider_Extend TO Dummy
  := SlidingCylinder.Extended;
END_TRANSITION
STEP Dummy:
END_STEP
TRANSITION FROM Dummy TO WP_Stamped
  := Check_Stamp_WPAvailable;
END_TRANSITION
STEP WP_Stamped:
  WPStamped(S);
  IsStamping(R);
END_STEP
TRANSITION FROM WP_Stamped TO Stamp_ACT_Stamp
  := WPStamped;
END_TRANSITION
END_ACTION

ACTION ACT_AutomaticExecute:
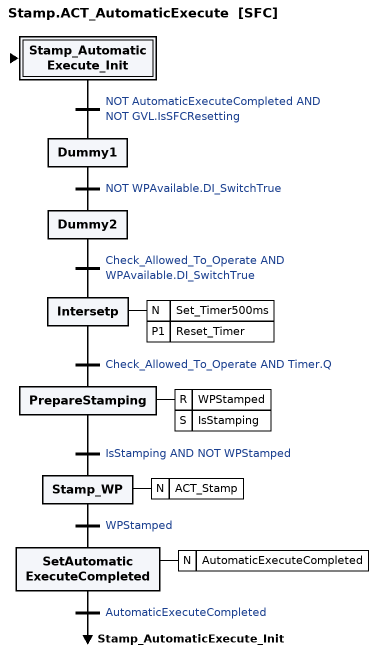
INITIAL_STEP Stamp_AutomaticExecute_Init:
END_STEP
TRANSITION FROM Stamp_AutomaticExecute_Init TO Dummy1
  := NOT AutomaticExecuteCompleted AND NOT GVL.IsSFCResetting;
END_TRANSITION
STEP Dummy1:
END_STEP
TRANSITION FROM Dummy1 TO Dummy2
  := NOT WPAvailable.DI_SwitchTrue;
END_TRANSITION
STEP Dummy2:
END_STEP
TRANSITION FROM Dummy2 TO Intersetp
  := Check_Allowed_To_Operate AND WPAvailable.DI_SwitchTrue;
END_TRANSITION
STEP Intersetp:
  Set_Timer500ms(N);
  Reset_Timer(P1);
END_STEP
TRANSITION FROM Intersetp TO PrepareStamping
  := Check_Allowed_To_Operate AND Timer.Q;
END_TRANSITION
STEP PrepareStamping:
  WPStamped(R);
  IsStamping(S);
END_STEP
TRANSITION FROM PrepareStamping TO Stamp_WP
  := IsStamping AND NOT WPStamped;
END_TRANSITION
STEP Stamp_WP:
  ACT_Stamp(N);
END_STEP
TRANSITION FROM Stamp_WP TO SetAutomaticExecuteCompleted
  := WPStamped;
END_TRANSITION
STEP SetAutomaticExecuteCompleted:
  AutomaticExecuteCompleted(N);
END_STEP
TRANSITION FROM SetAutomaticExecuteCompleted TO Stamp_AutomaticExecute_Init
  := AutomaticExecuteCompleted;
END_TRANSITION
END_ACTION

ACTION ACT_EmergencyStop:
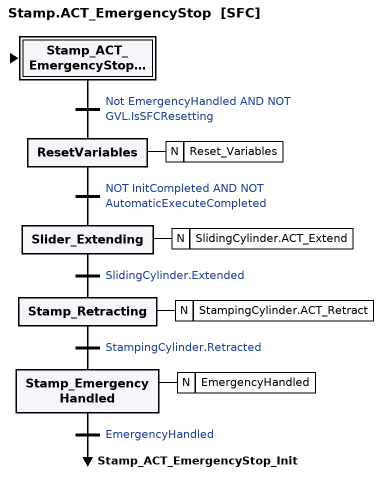
INITIAL_STEP Stamp_ACT_EmergencyStop_Init:
END_STEP
TRANSITION FROM Stamp_ACT_EmergencyStop_Init TO ResetVariables
  := Not EmergencyHandled AND NOT GVL.IsSFCResetting;
END_TRANSITION
STEP ResetVariables:
  Reset_Variables(N);
END_STEP
TRANSITION FROM ResetVariables TO Slider_Extending
  := NOT InitCompleted AND NOT AutomaticExecuteCompleted;
END_TRANSITION
STEP Slider_Extending:
  SlidingCylinder.ACT_Extend(N);
END_STEP
TRANSITION FROM Slider_Extending TO Stamp_Retracting
  := SlidingCylinder.Extended;
END_TRANSITION
STEP Stamp_Retracting:
  StampingCylinder.ACT_Retract(N);
END_STEP
TRANSITION FROM Stamp_Retracting TO Stamp_EmergencyHandled
  := StampingCylinder.Retracted;
END_TRANSITION
STEP Stamp_EmergencyHandled:
  EmergencyHandled(N);
END_STEP
TRANSITION FROM Stamp_EmergencyHandled TO Stamp_ACT_EmergencyStop_Init
  := EmergencyHandled;
END_TRANSITION
END_ACTION

ACTION ACT_Init:
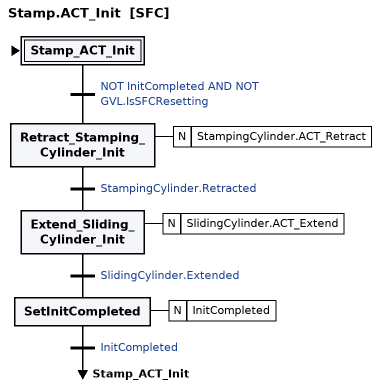
INITIAL_STEP Stamp_ACT_Init:
END_STEP
TRANSITION FROM Stamp_ACT_Init TO Retract_Stamping_Cylinder_Init
  := NOT InitCompleted AND NOT GVL.IsSFCResetting;
END_TRANSITION
STEP Retract_Stamping_Cylinder_Init:
  StampingCylinder.ACT_Retract(N);
END_STEP
TRANSITION FROM Retract_Stamping_Cylinder_Init TO Extend_Sliding_Cylinder_Init
  := StampingCylinder.Retracted;
END_TRANSITION
STEP Extend_Sliding_Cylinder_Init:
  SlidingCylinder.ACT_Extend(N);
END_STEP
TRANSITION FROM Extend_Sliding_Cylinder_Init TO SetInitCompleted
  := SlidingCylinder.Extended;
END_TRANSITION
STEP SetInitCompleted:
  InitCompleted(N);
END_STEP
TRANSITION FROM SetInitCompleted TO Stamp_ACT_Init
  := InitCompleted;
END_TRANSITION
END_ACTION
END_FUNCTION_BLOCK

FUNCTION_BLOCK PPU
                                            VAR_INPUT
                                            //Hardware
                                            Stack : Stack;
                                            Crane : Crane;
                                            Stamp : Stamp;
                                            //Software
                                            SFCReset : BOOL; //Only for SFC implementation
                                            END_VAR
                                            VAR_OUTPUT
                                            //Software
                                            StartButton : BOOL;
                                            InitCompleted : BOOL;
                                            AutomaticExecuteCompleted : BOOL;
                                            EmergencyStop : BOOL;
                                            EmergencyHandled : BOOL;
                                            SFCResetResetCompleted : BOOL; //Only for SFC implementation
                                            SFCResetCompleted : BOOL; //Only for SFC implementation
                                            END_VAR
                                            VAR
                                            END_VAR

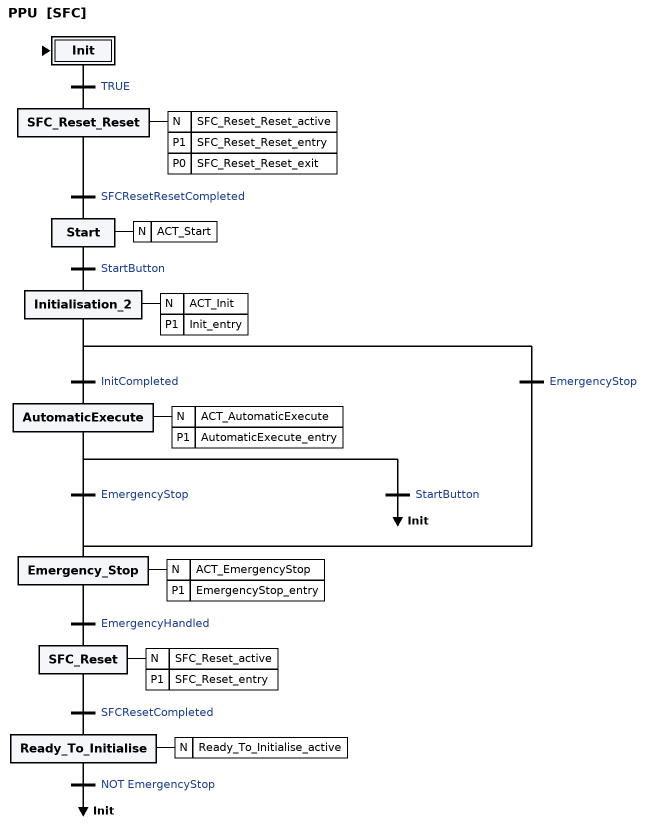
INITIAL_STEP Init:
END_STEP
TRANSITION FROM Init TO SFC_Reset_Reset
  := TRUE;
END_TRANSITION
STEP SFC_Reset_Reset:
  SFC_Reset_Reset_active(N);
  SFC_Reset_Reset_entry(P1);
  SFC_Reset_Reset_exit(P0);
END_STEP
TRANSITION FROM SFC_Reset_Reset TO Start
  := SFCResetResetCompleted;
END_TRANSITION
STEP Start:
  ACT_Start(N);
END_STEP
TRANSITION FROM Start TO Initialisation_2
  := StartButton;
END_TRANSITION
STEP Initialisation_2:
  ACT_Init(N);
  Init_entry(P1);
END_STEP
TRANSITION FROM Initialisation_2 TO AutomaticExecute
  := InitCompleted;
END_TRANSITION
TRANSITION FROM Initialisation_2 TO Emergency_Stop
  := EmergencyStop;
END_TRANSITION
STEP AutomaticExecute:
  ACT_AutomaticExecute(N);
  AutomaticExecute_entry(P1);
END_STEP
TRANSITION FROM AutomaticExecute TO Emergency_Stop
  := EmergencyStop;
END_TRANSITION
TRANSITION FROM AutomaticExecute TO Init
  := StartButton;
END_TRANSITION
STEP Emergency_Stop:
  ACT_EmergencyStop(N);
  EmergencyStop_entry(P1);
END_STEP
TRANSITION FROM Emergency_Stop TO SFC_Reset
  := EmergencyHandled;
END_TRANSITION
STEP SFC_Reset:
  SFC_Reset_active(N);
  SFC_Reset_entry(P1);
END_STEP
TRANSITION FROM SFC_Reset TO Ready_To_Initialise
  := SFCResetCompleted;
END_TRANSITION
STEP Ready_To_Initialise:
  Ready_To_Initialise_active(N);
END_STEP
TRANSITION FROM Ready_To_Initialise TO Init
  := NOT EmergencyStop;
END_TRANSITION

ACTION ACT_CheckEmergency:
                                            EmergencyStop :=
                                                Stack.EmergencyStop OR Stamp.EmergencyStop OR Crane.SoftwareEmergency OR
                                                Stamp.SoftwareEmergency;
                                            
                                        
END_ACTION

ACTION ACT_Start:
                                            StartButton := Stack.StartButton
                                                OR Stamp.StartButton;
                                            
                                        
END_ACTION

ACTION AutomaticExecute_entry:
                                            
                                                AutomaticExecuteCompleted:=FALSE;

                                                Stack.Panel.ACT_TurnLampWhite_Off();
                                                Stamp.Panel.ACT_TurnLampWhite_Off();
                                                Stack.Panel.ACT_TurnLampGreen_On();
                                                Stamp.Panel.ACT_TurnLampGreen_On();
                                            
                                        
END_ACTION

ACTION CallAll_AutomationExecutes:
                                            EmergencyStop :=
                                                Stack.EmergencyStop OR Stamp.EmergencyStop OR Crane.SoftwareEmergency OR
                                                Stamp.SoftwareEmergency;
                                                StartButton := Stack.StartButton OR Stamp.StartButton;
                                                Crane.ACT_AutomaticExecute();
                                                Stack.ACT_AutomaticExecute();
                                                Stamp.ACT_AutomaticExecute();
                                            
                                        
END_ACTION

ACTION EmergencyStop_entry:
                                            EmergencyHandled:=FALSE;

                                                Stack.Panel.ACT_TurnLampWhite_Off();
                                                Stamp.Panel.ACT_TurnLampWhite_Off();
                                                Stack.Panel.ACT_TurnLampGreen_Off();
                                                Stamp.Panel.ACT_TurnLampGreen_Off();
                                            
                                        
END_ACTION

ACTION Init_entry:
                                            InitCompleted:=FALSE;

                                                Stack.Panel.ACT_TurnLampWhite_On();
                                                Stamp.Panel.ACT_TurnLampWhite_On();
                                                Stack.Panel.ACT_TurnLampGreen_Off();
                                                Stamp.Panel.ACT_TurnLampGreen_Off();
                                            
                                        
END_ACTION

ACTION Ready_To_Initialise_active:
                                            EmergencyStop :=
                                                Stack.EmergencyStop OR Stamp.EmergencyStop OR Crane.SoftwareEmergency OR
                                                Stamp.SoftwareEmergency;
                                                StartButton := Stack.StartButton OR Stamp.StartButton;
                                                IF(StartButton)THEN
                                                Stamp.SoftwareEmergency:=FALSE;
                                                Crane.SoftwareEmergency:=FALSE;
                                                END_IF
                                            
                                        
END_ACTION

ACTION SFC_Reset_active:
                                            (*PPU*)
                                                //Variables
                                                InitCompleted:=FALSE;
                                                AutomaticExecuteCompleted:=FALSE;

                                                (*Crane Reset*)
                                                Crane(SFCReset:=TRUE);
                                                Crane.ACT_Init(SFCReset:=TRUE);
                                                Crane.ACT_AutomaticExecute(SFCReset:=TRUE);
                                                Crane.ACT_EmergencyStop(SFCReset:=TRUE);
                                                Crane.ACT_MoveToRamp(SFCReset:=TRUE);
                                                Crane.ACT_MoveToStack(SFCReset:=TRUE);
                                                Crane.ACT_MoveToStamp(SFCReset:=TRUE);
                                                Crane.ACT_PickUpWP(SFCReset:=TRUE);
                                                Crane.ACT_PutDownWP(SFCReset:=TRUE);

                                                (*Stack Reset*)
                                                Stack(SFCReset:=TRUE);
                                                Stack.ACT_Init(SFCReset:=TRUE);
                                                Stack.ACT_AutomaticExecute(SFCReset:=TRUE);
                                                Stack.ACT_ProvideWP(SFCReset:=TRUE);

                                                (*Stamp Reset*)
                                                Stamp(SFCReset:=TRUE);
                                                Stamp.ACT_Init(SFCReset:=TRUE);
                                                Stamp.ACT_AutomaticExecute(SFCReset:=TRUE);
                                                Stamp.ACT_Stamp(SFCReset:=TRUE);

                                                SFCResetCompleted:=TRUE;
                                            
                                        
END_ACTION

ACTION SFC_Reset_entry:
                                            SFCResetCompleted:=FALSE;
                                                GVL.IsSFCResetting:=TRUE;
                                            
                                        
END_ACTION

ACTION SFC_Reset_Reset_active:
                                            (*Crane Reset*)
                                                Crane(SFCReset:=FALSE);
                                                Crane.ACT_Init(SFCReset:=FALSE);
                                                Crane.ACT_AutomaticExecute(SFCReset:=FALSE);
                                                Crane.ACT_EmergencyStop(SFCReset:=FALSE);
                                                Crane.ACT_MoveToRamp(SFCReset:=FALSE);
                                                Crane.ACT_MoveToStack(SFCReset:=FALSE);
                                                Crane.ACT_MoveToStamp(SFCReset:=FALSE);
                                                Crane.ACT_PickUpWP(SFCReset:=FALSE);
                                                Crane.ACT_PutDownWP(SFCReset:=FALSE);
                                                Crane.LiftingCylinder.ACT_Retract();
                                                Crane.Gripper.ACT_Release();
                                                Crane.Table.Motor.ACT_Stop();
                                                //Variables
                                                Crane.InitCompleted:=FALSE;
                                                Crane.AutomaticExecuteCompleted:=FALSE;
                                                Crane.Stamp_AllowedToOperate:=FALSE;
                                                Crane.SoftwareEmergency:=FALSE;
                                                Crane.EmergencyHandled:=FALSE;
                                                Crane.SFCReset:=FALSE;

                                                (*Stack Reset*)
                                                Stack(SFCReset:=FALSE);
                                                Stack.ACT_Init(SFCReset:=FALSE);
                                                Stack.ACT_AutomaticExecute(SFCReset:=FALSE);
                                                Stack.ACT_ProvideWP(SFCReset:=FALSE);
                                                Stack.Seperator.ACT_Retract();
                                                //Variables
                                                Stack.InitCompleted:=FALSE;
                                                Stack.AutomaticExecuteCompleted:=FALSE;
                                                Stack.EmergencyHandled:=FALSE;
                                                Stack.SFCReset:=FALSE;

                                                (*Stamp Reset*)
                                                Stamp(SFCReset:=FALSE);
                                                Stamp.ACT_Init(SFCReset:=FALSE);
                                                Stamp.ACT_AutomaticExecute(SFCReset:=FALSE);
                                                Stamp.ACT_Stamp(SFCReset:=FALSE);
                                                Stamp.StampingCylinder.ACT_Retract();
                                                Stamp.SlidingCylinder.ACT_Extend();
                                                //Variables
                                                Stamp.InitCompleted:=FALSE;
                                                Stamp.AutomaticExecuteCompleted:=FALSE;
                                                Stamp.EmergencyHandled:=FALSE;
                                                Stamp.SFCReset:=FALSE;

                                                SFCResetResetCompleted:=TRUE;
                                                SFCResetCompleted:=TRUE;
                                            
                                        
END_ACTION

ACTION SFC_Reset_Reset_entry:
                                            SFCResetResetCompleted:=FALSE;
                                                GVL.IsSFCResetting:=TRUE;
                                            
                                        
END_ACTION

ACTION SFC_Reset_Reset_exit:
                                            GVL.IsSFCResetting:=FALSE;
                                            
                                        
END_ACTION

ACTION ACT_AutomaticExecute:
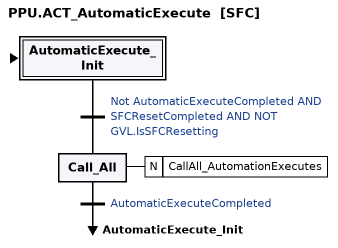
INITIAL_STEP AutomaticExecute_Init:
END_STEP
TRANSITION FROM AutomaticExecute_Init TO Call_All
  := Not AutomaticExecuteCompleted AND SFCResetCompleted AND NOT
                                                    GVL.IsSFCResetting;
END_TRANSITION
STEP Call_All:
  CallAll_AutomationExecutes(N);
END_STEP
TRANSITION FROM Call_All TO AutomaticExecute_Init
  := AutomaticExecuteCompleted;
END_TRANSITION
END_ACTION

ACTION ACT_EmergencyStop:
